// TwinCAT 3 PLC project PLC
// ProgramVersion: 3.1.4023.0
// libraries:
//   Tc2_Standard, * (Beckhoff Automation GmbH)
//   Tc2_System, * (Beckhoff Automation GmbH)
//   Tc3_Module, * (Beckhoff Automation GmbH)
// project tree:
//   GVLs/ GVL.TcGVL
//   / PlcTask.TcTTO (not stored)
//   POUs/Actuators/ Contactor.TcPOU, DirectOnlineStarterMotor.TcPOU, I_SingleDirectionMotor.TcIO (not stored)
//   POUs/Devices/ I_PushButton.TcIO, I_Sensor.TcIO (not stored), NormallyClosedSensor.TcPOU, NormallyOpenPushButton.TcPOU, NormallyClosedPushButton.TcPOU, NormallyOpenSensor.TcPOU
//   POUs/Machines/ ConveyorSortingMachine.TcPOU
//   POUs/ MAIN.TcPOU
//   POUs/Modules/ I_Module.TcIO (not stored), SortingConveyor.TcPOU
// real-time tasks:
//   TASK PlcTask: cycle T#10ms, priority 20, ADS port 350
//   TASK PlcTask1: cycle T#10ms, priority 21, ADS port 351
//   TASK PlcTask2: cycle T#10ms, priority 22, ADS port 352

// ---- GVLs/GVL.TcGVL
{attribute 'qualified_only'}
VAR_GLOBAL
	emergencyStopButton				: NormallyClosedPushButton;
	stopButton						: NormallyClosedPushButton;
	startButton						: NormallyOpenPushButton;
	
	productDetectedSensor			: NormallyClosedSensor;
	conveyorFullSensor				: NormallyClosedSensor;

	conveyorMotor					: DirectOnlineStarterMotor;
	
	sortingConveyor					: SortingConveyor(
										productDetected		:= productDetectedSensor,
										conveyorFull		:= conveyorFullSensor,
										conveyor			:= conveyorMotor);
	
	myConveyorSortingMachine		: ConveyorSortingMachine(
										emergencyStopButton	:= emergencyStopButton,
										stopButton			:= stopButton,
										startButton			:= startButton,	
										conveyorModule		:= sortingCOnveyor);
	
	
END_VAR

// ---- POUs/Devices/I_PushButton.TcIO
INTERFACE I_PushButton

PROPERTY IsPressed : Bool
GET
END_GET
END_PROPERTY

PROPERTY IsReleased : Bool
GET
END_GET
END_PROPERTY

END_INTERFACE

// ---- POUs/Devices/NormallyClosedPushButton.TcPOU
{attribute 'no_explicit_call' := 'NormallyClosedPushButton is a CLASS and must be accessed using methods or properties'}
FUNCTION_BLOCK NormallyClosedPushButton implements I_PushButton
VAR
	input				AT %I*: BOOL;
END_VAR

PROPERTY IsPressed : bool
GET
IsPressed				:= not input;
END_GET
END_PROPERTY

PROPERTY IsReleased : bool
GET
IsReleased				:= input;
END_GET
END_PROPERTY

END_FUNCTION_BLOCK

// ---- POUs/Devices/NormallyOpenPushButton.TcPOU
{attribute 'no_explicit_call' := 'NormallyOpenPushButton is a CLASS and must be accessed using methods or properties'}
FUNCTION_BLOCK NormallyOpenPushButton
VAR
	input				AT %I*: BOOL;
END_VAR

PROPERTY IsPressed : bool
GET
IsPressed				:= input;
END_GET
END_PROPERTY

PROPERTY IsReleased : bool
GET
IsPressed				:= not input;
END_GET
END_PROPERTY

END_FUNCTION_BLOCK

// ---- POUs/Devices/NormallyClosedSensor.TcPOU
{attribute 'no_explicit_call' := 'NormallyClosedSensor is a CLASS and must be accessed using methods or properties'}
FUNCTION_BLOCK NormallyClosedSensor
VAR
	input				AT %I*: BOOL;
END_VAR

PROPERTY IsActive : bool
GET
IsActive				:= input;
END_GET
END_PROPERTY

PROPERTY IsNotActive : bool
GET
IsActive				:= not input;
END_GET
END_PROPERTY

END_FUNCTION_BLOCK

// ---- POUs/Actuators/DirectOnlineStarterMotor.TcPOU
{attribute 'no_explicit_call' := 'DriectOnlineStarterMotor is a CLASS and must be accessed using methods or properties'}
FUNCTION_BLOCK DirectOnlineStarterMotor implements I_SingleDirectionMotor
VAR
	contactor			: Contactor;
END_VAR

METHOD Start
contactor.SwitchOn();
END_METHOD

METHOD Stop
contactor.SwitchOff();
END_METHOD

END_FUNCTION_BLOCK

// ---- POUs/Actuators/Contactor.TcPOU
{attribute 'no_explicit_call' := 'Contactor is a CLASS and must be accessed using methods or properties'}
FUNCTION_BLOCK Contactor
VAR
	output				AT %Q*: BOOL;
END_VAR

METHOD SwitchOff
VAR_INPUT
END_VAR
output   := false;
END_METHOD

METHOD SwitchOn
VAR_INPUT
END_VAR
output   := true;
END_METHOD

END_FUNCTION_BLOCK

// ---- POUs/Modules/SortingConveyor.TcPOU
FUNCTION_BLOCK SortingConveyor IMPLEMENTS I_Module
VAR
	productDetected			: I_Sensor;
	conveyorFull			: I_Sensor;
	conveyor				: I_SingleDirectionMotor;
	enabled					: BOOL;
	timeout					: tof;
END_VAR

// Minimum time the conveyor keeps on running
Timeout(IN:= enabled AND productDetected.IsActive, PT:=T#5S, Q=> , ET=> );
// Conveyor keeps on running until not full and some extra time
IF enabled AND Timeout.Q AND conveyorFull.IsNotActive THEN
	conveyor.Start();
ELSE
	conveyor.Stop();
END_IF

{warning 'add method implementation '}
METHOD Disable
enabled := false;
END_METHOD

{warning 'add method implementation '}
METHOD Enable
enabled := true;
END_METHOD

METHOD FB_init : BOOL
VAR_INPUT
	bInitRetains : BOOL; // if TRUE, the retain variables are initialized (warm start / cold start)
	bInCopyCode : BOOL;  // if TRUE, the instance afterwards gets moved into the copy code (online change)
	productDetected			: I_Sensor;
	conveyorFull			: I_Sensor;
	conveyor				: I_SingleDirectionMotor;
END_VAR
THIS^.productDetected		:= productDetected;
THIS^.conveyorFull			:= conveyorFull;
THIS^.conveyor				:= conveyor;
END_METHOD

END_FUNCTION_BLOCK

// ---- POUs/Machines/ConveyorSortingMachine.TcPOU
FUNCTION_BLOCK ConveyorSortingMachine
VAR
	emergencyStopButton				: I_PushButton;
	stopButton						: I_PushButton;
	startButton						: I_PushButton;	
	conveyorModule					: I_Module;
END_VAR

// Conveyor control is ok when the ES nor the stop button is pushed
IF StopButton.IsPressed OR EmergencyStopButton.IsPressed	THEN
	conveyorModule.Disable();
	
ELSIF StartButton.IsPressed	AND StopButton.IsReleased		THEN
	conveyorModule.Enable();	
	
END_IF

METHOD FB_init : BOOL
VAR_INPUT
	bInitRetains : BOOL; // if TRUE, the retain variables are initialized (warm start / cold start)
	bInCopyCode : BOOL;  // if TRUE, the instance afterwards gets moved into the copy code (online change)
	emergencyStopButton				: I_PushButton;
	stopButton						: I_PushButton;
	startButton						: I_PushButton;	
	conveyorModule					: I_Module;
END_VAR
THIS^.emergencyStopButton				:= emergencyStopButton;
THIS^.stopButton						:= stopButton;
THIS^.startButton						:= startButton;	
THIS^.conveyorModule					:= conveyorModule;
END_METHOD

END_FUNCTION_BLOCK

// ---- POUs/Devices/NormallyOpenSensor.TcPOU
{attribute 'no_explicit_call' := 'NormallyOpenSensor is a CLASS and must be accessed using methods or properties'}
FUNCTION_BLOCK NormallyOpenSensor implements I_Sensor
VAR
	input				AT %I*: BOOL;
END_VAR

PROPERTY IsActive : bool
GET
IsActive				:= not input;
END_GET
END_PROPERTY

PROPERTY IsNotActive : bool
GET
IsActive				:= input;
END_GET
END_PROPERTY

END_FUNCTION_BLOCK

// ---- POUs/MAIN.TcPOU
PROGRAM MAIN
VAR
	ConveyorControl				: BOOL;
	Timeout						: TOF;
END_VAR

// Conveyor control is ok when the ES nor the stop button is pushed
IF GVL.StopButton.IsPressed OR GVL.EmergencyStopButton.IsPressed	THEN
	ConveyorControl	:= FALSE;
	
ELSIF gvl.StartButton.IsPressed	AND gvl.StopButton.IsReleased		THEN
	ConveyorControl	:= TRUE;
	
END_IF

// Minimum time the conveyor keeps on running
Timeout(IN:= ConveyorControl AND gvl.ProductDetectedSensor.IsActive, PT:=T#5S, Q=> , ET=> );
// Conveyor keeps on running until not full and some extra time
gvl.MotorContactor	:= ConveyorControl AND Timeout.Q AND NOT gvl.ConveyorFullSensor;

END_PROGRAM
